{attribute 'qualified_only'}
TYPE E_WFS_States :
(
    Unknown := 0,
    OUT := 1,
    TARGET1 := 2,
    TARGET2 := 3,
    TARGET3 := 4,
    TARGET4 := 5,
    TARGET5 := 6
) UINT;
END_TYPE

(* stored: Version 1.1.0.1
   DUT E_WFS_States: Id {3453a453-2671-4525-8745-914037e14ff2} *)
